TYPE "Prod_Beam_Data"
VERSION : 0.1
// Block: Prod_Beam_Data
   STRUCT
      O_ACT : Prod_Item_small;
      O_TODO : Array[1..15] of Prod_Item_small;
      O_ENDING : Array[1..5] of Prod_Item_small;
      O_OUT : Array[1..5] of Prod_Item_small;
   END_STRUCT;

END_TYPE
